FUNCTION TryConvert_DWORD_TO_UDINT : BOOL
VAR_INPUT
	in : DWORD;
	out : REFERENCE TO UDINT;
END_VAR

out := DWORD_TO_UDINT(in);
TryConvert_DWORD_TO_UDINT := TRUE;

END_FUNCTION

(* stored: Version 1.1.0.1, ProductVersion 3.1.4024.12
   POU TryConvert_DWORD_TO_UDINT: Id {14f1b7b9-d4d1-4ae9-bf68-a3fe9a88e820}, SpecialFunc None *)
